Universal Robots PolyScope program: test.urp

Program test (installation=default directory=/programs/usbdisk createdIn=3.8.0.61336 lastSavedIn=3.8.0.61336 robotSerialNumber=2017355926)
Calibrated DH parameters: a=[0.000209, -0.089833, -0.171809, 0.000042, 0.00009, 0]; d=[0.089446, 227.121722, -1643.006454, 1415.994937, 0.094815, 0.082468]; alpha=[1.569174, -0.001831, 0.000249, 1.569946, -1.570307, 0]; deltaTheta=[-0.000025, -1.358049, 0.240417, 1.117537, -0.00004, 0.000045]
Robot Program (runOnlyOnce=false)
  MoveJ speed 60 deg/s, acceleration 80 deg/s^2 (useActiveTCP=true)
    Waypoint Waypoint_1: TCP in base x=0.259 y=-509.462 z=601.133 mm, rx=0.0007 ry=-2.2217 rz=2.221 rad; joints [-4.646, -50.897, -84.316, 134.216, -4.572, -179.02] deg; flange x=0.182 y=-192.462 z=601.236 mm, rx=0.0007 ry=-2.2217 rz=2.221 rad
  Wait Sleep waitTime=2
  MoveJ speed 60 deg/s, acceleration 80 deg/s^2 (useActiveTCP=true)
    Waypoint Waypoint_2: TCP in base x=0.207 y=-509.46 z=1001.928 mm, rx=0.0003 ry=-2.2218 rz=2.2211 rad; joints [-0.003, -90.002, 0.002, -90.003, -0.002, -0.003] deg; flange x=0.166 y=-192.46 z=1002.024 mm, rx=0.0003 ry=-2.2218 rz=2.2211 rad
  Wait Sleep waitTime=2
